INTERFACE I_ActuatorPosNeg EXTENDS I_ActuatorBase

{attribute 'monitoring' := 'call'}
PROPERTY public negativeOk : BOOL
GET
END_GET
END_PROPERTY

METHOD PUBLIC negativeOn : BOOL
VAR_INPUT
END_VAR
END_METHOD

{attribute 'monitoring' := 'call'}
PROPERTY public positiveOk : BOOL
GET
END_GET
END_PROPERTY

METHOD PUBLIC positiveOn : BOOL
VAR_INPUT
END_VAR
END_METHOD

END_INTERFACE

(* stored: Version 1.1.0.1, ProductVersion 3.1.4024.3
   Itf I_ActuatorPosNeg: Id {c1cd79fb-ef10-4df4-a967-a7af4ba9ed11}
   Property negativeOk: Id {acaaf001-24c3-49e1-a0b0-ae4d3cb97674}
   Get Get: Id {64c8668d-5829-4441-8bdf-4cc05643fa43}
   Method negativeOn: Id {52c08776-8aa9-41d5-92fc-8e4de4251cdf}
   Property positiveOk: Id {c368d4ad-cb52-4aac-9776-e44d44da6954}
   Get Get: Id {3a19b69a-56a6-4b5b-ab7b-7a647caed44d}
   Method positiveOn: Id {552a88d5-2c90-430d-ac56-c7f8d70f3f54} *)
